{attribute 'qualified_only'}
VAR_GLOBAL
	Fixture1Input:FixtureInput;
	Fixture1Output:FixtureOutput;
	Fixture2Input:FixtureInput;
	Fixture2Output:FixtureOutput;
END_VAR

(* stored: Version 1.1.0.1, ProductVersion 3.1.4024.16
   GVL IO: Id {c8116558-34ab-4d50-b878-244311207243} *)
